// Mitsubishi GX Works2 project: fx1s_ykhmi_thao may_230929   PLC: FX1S

PROGRAM MAIN
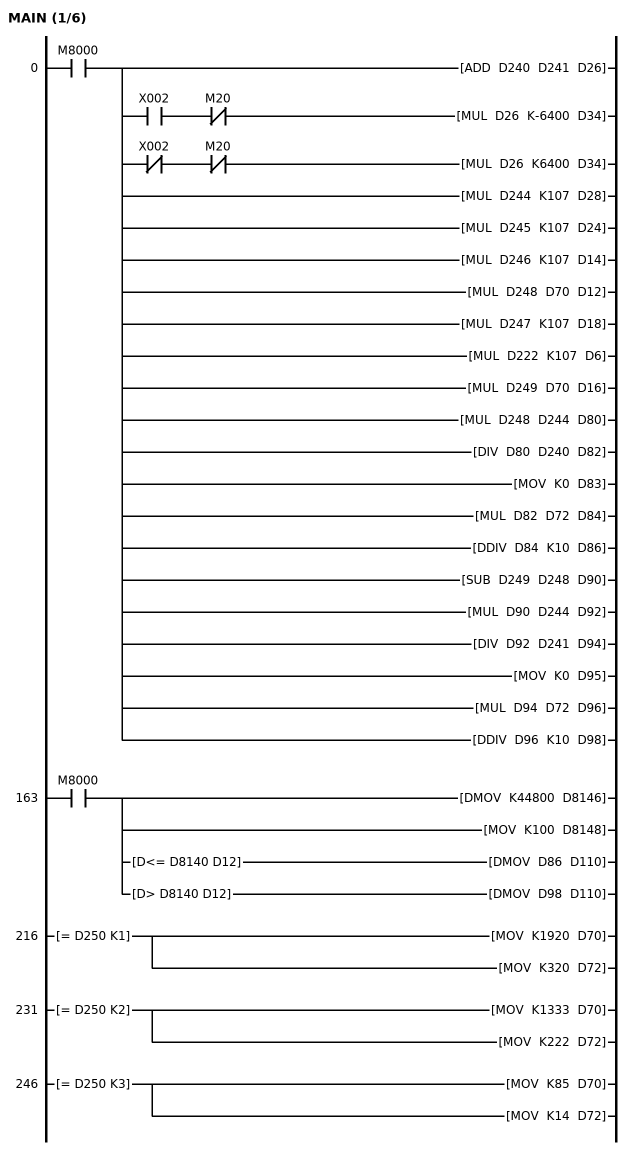
0     LD      M8000
      ADD     D240 D241 D26
      MPS
      AND     X002
      ANI     M20
      MUL     D26 K-6400 D34
      MRD
      ANI     X002
      ANI     M20
      MUL     D26 K6400 D34
      MPP
      MUL     D244 K107 D28
      MUL     D245 K107 D24
      MUL     D246 K107 D14
      MUL     D248 D70 D12
      MUL     D247 K107 D18
      MUL     D222 K107 D6
      MUL     D249 D70 D16
      MUL     D248 D244 D80
      DIV     D80 D240 D82
      MOV     K0 D83
      MUL     D82 D72 D84
      DDIV    D84 K10 D86
      SUB     D249 D248 D90
      MUL     D90 D244 D92
      DIV     D92 D241 D94
      MOV     K0 D95
      MUL     D94 D72 D96
      DDIV    D96 K10 D98
163   LD      M8000
      DMOV    K44800 D8146
      MOV     K100 D8148
      MPS
      ANDD<=  D8140 D12
      DMOV    D86 D110
      MPP
      ANDD>   D8140 D12
      DMOV    D98 D110
216   LD=     D250 K1
      MOV     K1920 D70
      MOV     K320 D72
231   LD=     D250 K2
      MOV     K1333 D70
      MOV     K222 D72
246   LD=     D250 K3
      MOV     K85 D70
      MOV     K14 D72
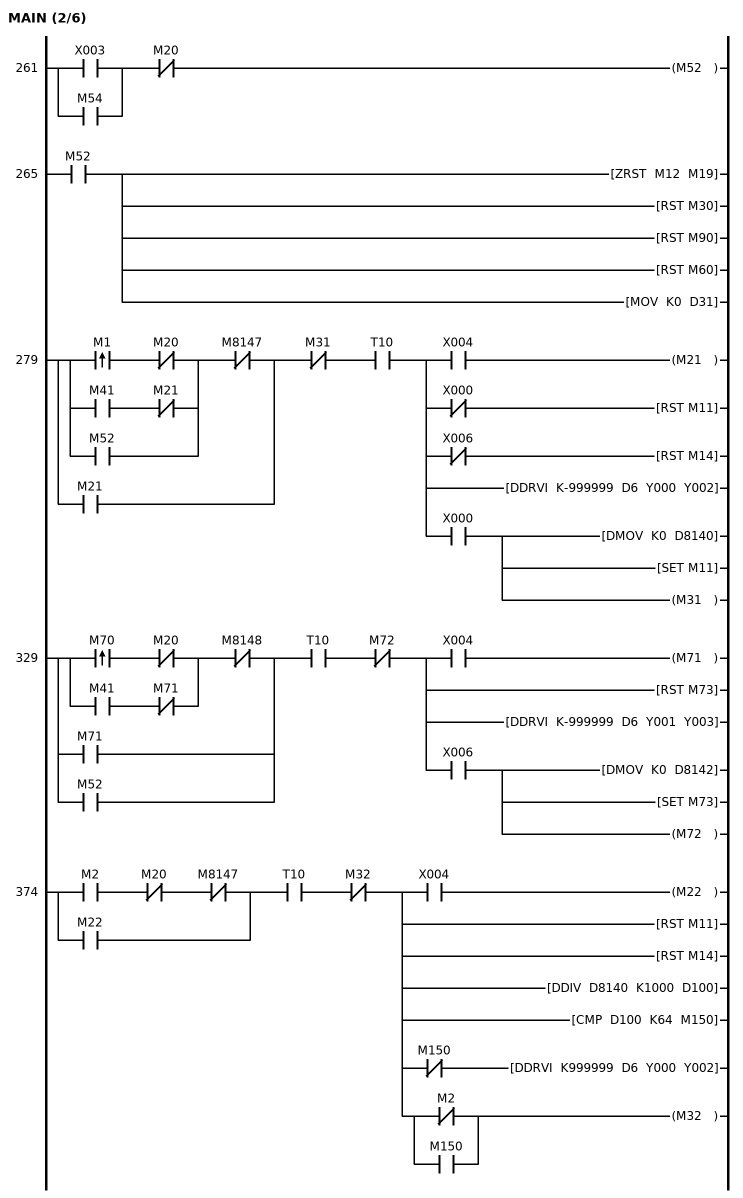
261   LD      X003
      OR      M54
      ANI     M20
      OUT     M52
265   LD      M52
      ZRST    M12 M19
      RST     M30
      RST     M90
      RST     M60
      MOV     K0 D31
279   LDP     M1
      ANI     M20
      LD      M41
      ANI     M21
      ORB
      OR      M52
      ANI     M8147
      OR      M21
      ANI     M31
      AND     T10
      MPS
      AND     X004
      OUT     M21
      MRD
      ANI     X000
      RST     M11
      MRD
      ANI     X006
      RST     M14
      MPP
      DDRVI   K-999999 D6 Y000 Y002
      AND     X000
      DMOV    K0 D8140
      SET     M11
      OUT     M31
329   LDP     M70
      ANI     M20
      LD      M41
      ANI     M71
      ORB
      ANI     M8148
      OR      M71
      OR      M52
      AND     T10
      ANI     M72
      MPS
      AND     X004
      OUT     M71
      MPP
      RST     M73
      DDRVI   K-999999 D6 Y001 Y003
      AND     X006
      DMOV    K0 D8142
      SET     M73
      OUT     M72
374   LD      M2
      ANI     M20
      ANI     M8147
      OR      M22
      AND     T10
      ANI     M32
      MPS
      AND     X004
      OUT     M22
      MPP
      RST     M11
      RST     M14
      DDIV    D8140 K1000 D100
      CMP     D100 K64 M150
      MPS
      ANI     M150
      DDRVI   K999999 D6 Y000 Y002
      MPP
      LDI     M2
      OR      M150
      ANB
      OUT     M32
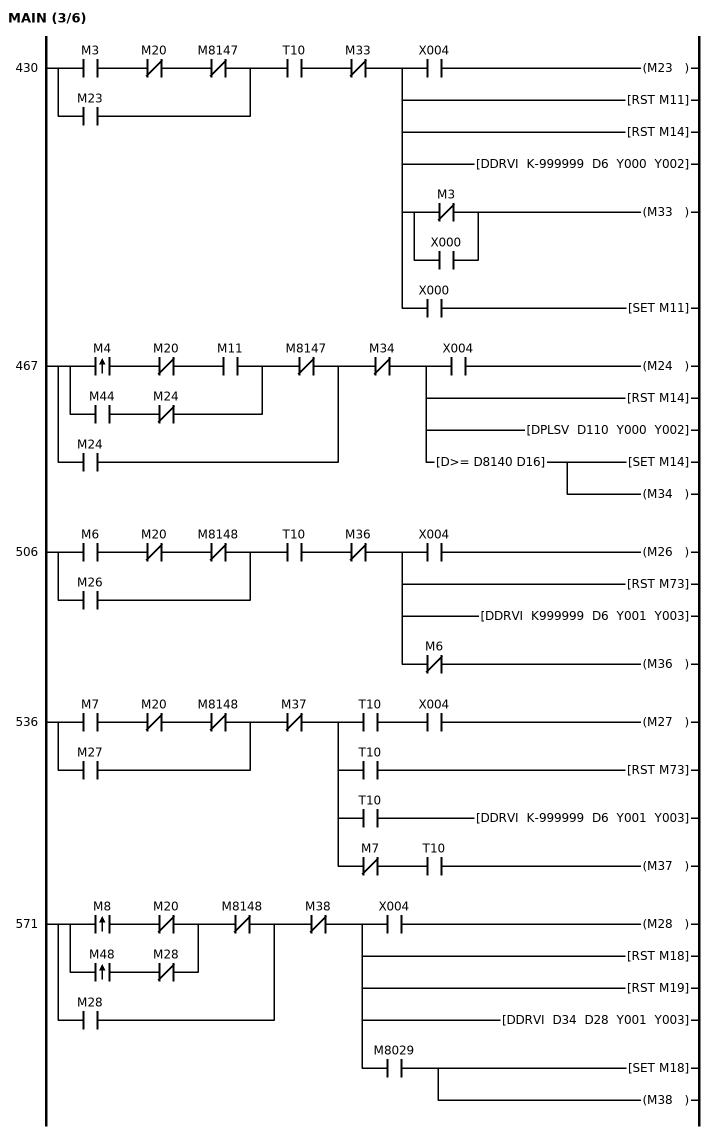
430   LD      M3
      ANI     M20
      ANI     M8147
      OR      M23
      AND     T10
      ANI     M33
      MPS
      AND     X004
      OUT     M23
      MPP
      RST     M11
      RST     M14
      DDRVI   K-999999 D6 Y000 Y002
      MPS
      LDI     M3
      OR      X000
      ANB
      OUT     M33
      MPP
      AND     X000
      SET     M11
467   LDP     M4
      ANI     M20
      AND     M11
      LD      M44
      ANI     M24
      ORB
      ANI     M8147
      OR      M24
      ANI     M34
      MPS
      AND     X004
      OUT     M24
      MPP
      RST     M14
      DPLSV   D110 Y000 Y002
      ANDD>=  D8140 D16
      SET     M14
      OUT     M34
506   LD      M6
      ANI     M20
      ANI     M8148
      OR      M26
      AND     T10
      ANI     M36
      MPS
      AND     X004
      OUT     M26
      MPP
      RST     M73
      DDRVI   K999999 D6 Y001 Y003
      ANI     M6
      OUT     M36
536   LD      M7
      ANI     M20
      ANI     M8148
      OR      M27
      ANI     M37
      MPS
      AND     T10
      AND     X004
      OUT     M27
      MRD
      AND     T10
      RST     M73
      MRD
      AND     T10
      DDRVI   K-999999 D6 Y001 Y003
      MPP
      ANI     M7
      AND     T10
      OUT     M37
571   LDP     M8
      ANI     M20
      LDP     M48
      ANI     M28
      ORB
      ANI     M8148
      OR      M28
      ANI     M38
      MPS
      AND     X004
      OUT     M28
      MPP
      RST     M18
      RST     M19
      DDRVI   D34 D28 Y001 Y003
      AND     M8029
      SET     M18
      OUT     M38
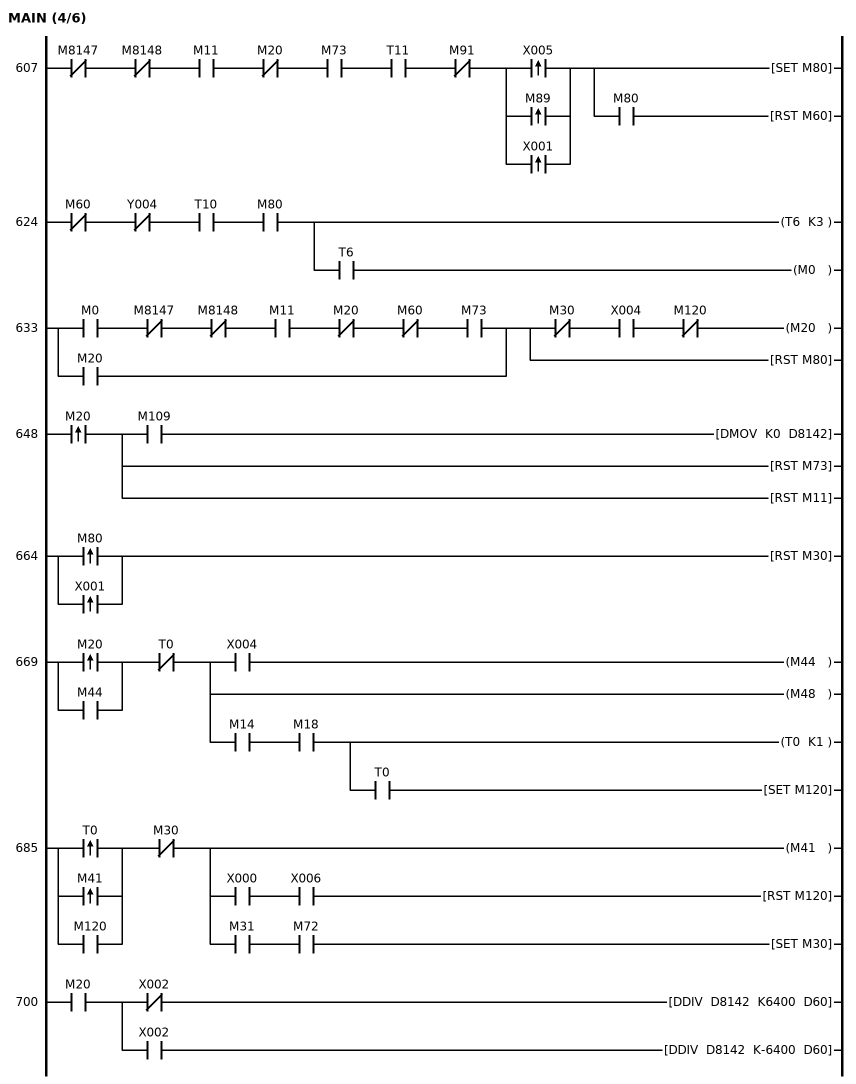
607   LDI     M8147
      ANI     M8148
      AND     M11
      ANI     M20
      AND     M73
      AND     T11
      ANI     M91
      LDP     X005
      ORP     M89
      ORP     X001
      ANB
      SET     M80
      AND     M80
      RST     M60
624   LDI     M60
      ANI     Y004
      AND     T10
      AND     M80
      OUT     T6 K3
      AND     T6
      OUT     M0
633   LD      M0
      ANI     M8147
      ANI     M8148
      AND     M11
      ANI     M20
      ANI     M60
      AND     M73
      OR      M20
      MPS
      ANI     M30
      AND     X004
      ANI     M120
      OUT     M20
      MPP
      RST     M80
648   LDP     M20
      MPS
      AND     M109
      DMOV    K0 D8142
      MPP
      RST     M73
      RST     M11
664   LDP     M80
      ORP     X001
      RST     M30
669   LDP     M20
      OR      M44
      ANI     T0
      MPS
      AND     X004
      OUT     M44
      MPP
      OUT     M48
      AND     M14
      AND     M18
      OUT     T0 K1
      AND     T0
      SET     M120
685   LDP     T0
      ORP     M41
      OR      M120
      ANI     M30
      OUT     M41
      MPS
      AND     X000
      AND     X006
      RST     M120
      MPP
      AND     M31
      AND     M72
      SET     M30
700   LD      M20
      MPS
      ANI     X002
      DDIV    D8142 K6400 D60
      MPP
      AND     X002
      DDIV    D8142 K-6400 D60
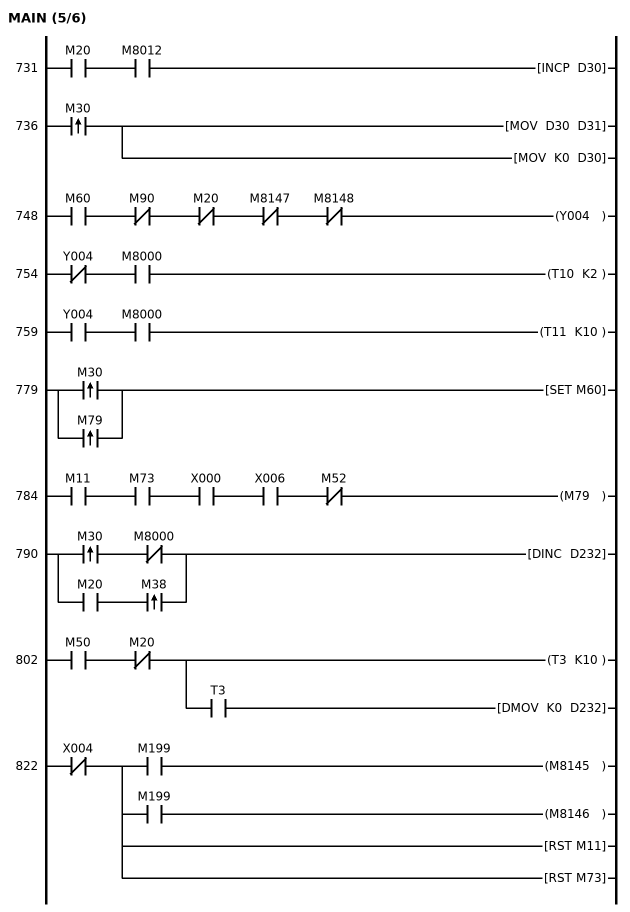
731   LD      M20
      AND     M8012
      INCP    D30
736   LDP     M30
      MOV     D30 D31
      MOV     K0 D30
748   LD      M60
      ANI     M90
      ANI     M20
      ANI     M8147
      ANI     M8148
      OUT     Y004
754   LDI     Y004
      AND     M8000
      OUT     T10 K2
759   LD      Y004
      AND     M8000
      OUT     T11 K10
779   LDP     M30
      ORP     M79
      SET     M60
784   LD      M11
      AND     M73
      AND     X000
      AND     X006
      ANI     M52
      OUT     M79
790   LDP     M30
      ANI     M8000
      LD      M20
      ANDP    M38
      ORB
      DINC    D232
802   LD      M50
      ANI     M20
      OUT     T3 K10
      AND     T3
      DMOV    K0 D232
822   LDI     X004
      MPS
      AND     M199
      OUT     M8145
      MRD
      AND     M199
      OUT     M8146
      MPP
      RST     M11
      RST     M73
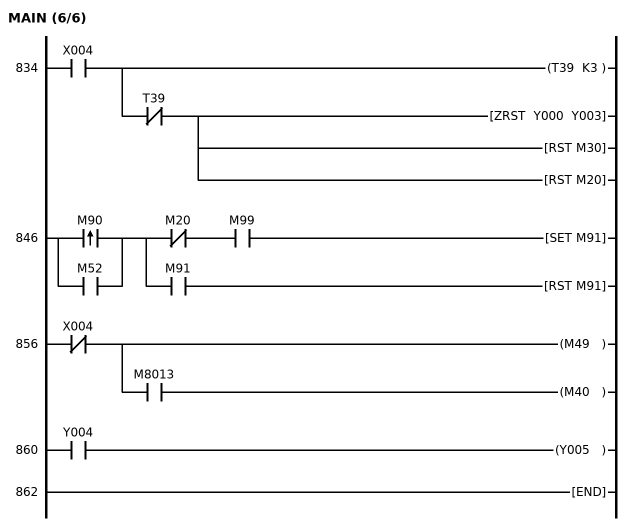
834   LD      X004
      OUT     T39 K3
      ANI     T39
      ZRST    Y000 Y003
      RST     M30
      RST     M20
846   LDP     M90
      OR      M52
      MPS
      ANI     M20
      AND     M99
      SET     M91
      MPP
      AND     M91
      RST     M91
856   LDI     X004
      OUT     M49
      AND     M8013
      OUT     M40
860   LD      Y004
      OUT     Y005
862   END
END_PROGRAM
